// TIA Portal V16 export
// export: Created 2024-12-03T15:41:45.1600688Z, ExportSetting WithReadOnly, DisplayName Totally Integrated Automation Portal, DisplayVersion V16 Update 6, DisplayName TIA Portal Version Control Interface, DisplayVersion V16 Update 2, DisplayName TIA Portal Openness, DisplayVersion V16 Update 6, DisplayName TIA Portal Teamcenter Gateway, DisplayVersion V16, DisplayName SINAMICS Startdrive Advanced, DisplayVersion V16 Update 5, DisplayName SINAMICS Startdrive G130, G150, S120, S150, SINAMICS MV, S210, DisplayVersion V16 Update 5, DisplayName SINAMICS Startdrive G110M, G120, G120C, G120D, G120P, G115D, DisplayVersion V16 Update 5, DisplayName STEP 7 Professional, DisplayVersion V16 Update 6, DisplayName STEP 7 Safety, DisplayVersion V16, DisplayName WinCC Advanced / Unified PC, DisplayVersion V16 Update 6
TYPE "IT2000M_Scale_OUT_UDT"
// stored: CreationDate 2021-07-13T07:41:36.2278727Z, InterfaceModifiedDate 2021-07-11T06:56:03.4179476Z, IsConsistent true, LibraryConformanceStatus The object is library-conformant., ModifiedDate 2021-07-11T06:56:03.4179476Z
   STRUCT
      Commands : Struct
         AbortFilling : Bool;
         AckOutOfTolerance : Bool;
         StopBeforeToleranceCheck : Bool;
         ShowText : Bool;
         SetDigitalOutputs : Bool;
         WeightStorage : Bool;
         spare_0 : Bool;
         spare_1 : Bool;
         SetZero : Bool;
         AutoTaring : Bool;
         SetToGross : Bool;
         ManualTaring : Bool;
         FillingWithoutTaring : Bool;
         StartFilling : Bool;
         StartDischarging : Bool;
         InterruptFilling : Bool;
      END_STRUCT;
      reserve : Word;
      TareValue : Int;
      TargetWeight : Int;
      PreactFast : Int;
      PreactSlow : Int;
      TolerancePos : Int;
      ToleranceNeg : Int;
      SettlingTimeMs : Int;
      JogPulseMs : Int;
      WeightDiffForFlowRateCheck : Int;
      TImeINtervalForFlowRateCheck : Int;
      ZeroRange : Int;
      ExtenedDischargingTimeMs : Int;
   END_STRUCT;
END_TYPE
